{attribute 'GeneratedUsingTerminal: APS4322-7000-0017'}
{attribute addProperty BoxType "APS4322-7000-0017"}
{attribute addProperty Id "StatusWordAT %I*UINT2Current_D_0X0AT %I*INT2Current_D_0X1AT %I*INT2Current_D_0X2AT %I*INT2Current_D_0Y0AT %I*INT2Current_D_0Y1AT %I*INT2Current_D_0Y2AT %I*INT2Current_D_1X0AT %I*INT2Current_D_1X1AT %I*INT2Current_D_1X2AT %I*INT2Current_D_1Y0AT %I*INT2Current_D_1Y1AT %I*INT2Current_D_1Y2AT %I*INT2Current_D_2X0AT %I*INT2Current_D_2X1AT %I*INT2Current_D_2X2AT %I*INT2Current_D_2Y0AT %I*INT2Current_D_2Y1AT %I*INT2Current_D_2Y2AT %I*INT2Current_D_3X0AT %I*INT2Current_D_3X1AT %I*INT2Current_D_3X2AT %I*INT2Current_D_3Y0AT %I*INT2Current_D_3Y1AT %I*INT2Current_D_3Y2AT %I*INT2Current_Q_0X0AT %I*INT2Current_Q_0X1AT %I*INT2Current_Q_0X2AT %I*INT2Current_Q_0Y0AT %I*INT2Current_Q_0Y1AT %I*INT2Current_Q_0Y2AT %I*INT2Current_Q_1X0AT %I*INT2Current_Q_1X1AT %I*INT2Current_Q_1X2AT %I*INT2Current_Q_1Y0AT %I*INT2Current_Q_1Y1AT %I*INT2Current_Q_1Y2AT %I*INT2Current_Q_2X0AT %I*INT2Current_Q_2X1AT %I*INT2Current_Q_2X2AT %I*INT2Current_Q_2Y0AT %I*INT2Current_Q_2Y1AT %I*INT2Current_Q_2Y2AT %I*INT2Current_Q_3X0AT %I*INT2Current_Q_3X1AT %I*INT2Current_Q_3X2AT %I*INT2Current_Q_3Y0AT %I*INT2Current_Q_3Y1AT %I*INT2Current_Q_3Y2AT %I*INT2"}
{attribute addProperty CRC "1192874203"}
{attribute addProperty Size "98"}
TYPE APS_Inputs_4719D0DB :
STRUCT
	{attribute addProperty Name "StatusWord"}
	StatusWord AT %I* : UINT;
	{attribute addProperty Name "Current_D_0X0"}
	Current_D_0X0 AT %I* : INT;
	{attribute addProperty Name "Current_D_0X1"}
	Current_D_0X1 AT %I* : INT;
	{attribute addProperty Name "Current_D_0X2"}
	Current_D_0X2 AT %I* : INT;
	{attribute addProperty Name "Current_D_0Y0"}
	Current_D_0Y0 AT %I* : INT;
	{attribute addProperty Name "Current_D_0Y1"}
	Current_D_0Y1 AT %I* : INT;
	{attribute addProperty Name "Current_D_0Y2"}
	Current_D_0Y2 AT %I* : INT;
	{attribute addProperty Name "Current_D_1X0"}
	Current_D_1X0 AT %I* : INT;
	{attribute addProperty Name "Current_D_1X1"}
	Current_D_1X1 AT %I* : INT;
	{attribute addProperty Name "Current_D_1X2"}
	Current_D_1X2 AT %I* : INT;
	{attribute addProperty Name "Current_D_1Y0"}
	Current_D_1Y0 AT %I* : INT;
	{attribute addProperty Name "Current_D_1Y1"}
	Current_D_1Y1 AT %I* : INT;
	{attribute addProperty Name "Current_D_1Y2"}
	Current_D_1Y2 AT %I* : INT;
	{attribute addProperty Name "Current_D_2X0"}
	Current_D_2X0 AT %I* : INT;
	{attribute addProperty Name "Current_D_2X1"}
	Current_D_2X1 AT %I* : INT;
	{attribute addProperty Name "Current_D_2X2"}
	Current_D_2X2 AT %I* : INT;
	{attribute addProperty Name "Current_D_2Y0"}
	Current_D_2Y0 AT %I* : INT;
	{attribute addProperty Name "Current_D_2Y1"}
	Current_D_2Y1 AT %I* : INT;
	{attribute addProperty Name "Current_D_2Y2"}
	Current_D_2Y2 AT %I* : INT;
	{attribute addProperty Name "Current_D_3X0"}
	Current_D_3X0 AT %I* : INT;
	{attribute addProperty Name "Current_D_3X1"}
	Current_D_3X1 AT %I* : INT;
	{attribute addProperty Name "Current_D_3X2"}
	Current_D_3X2 AT %I* : INT;
	{attribute addProperty Name "Current_D_3Y0"}
	Current_D_3Y0 AT %I* : INT;
	{attribute addProperty Name "Current_D_3Y1"}
	Current_D_3Y1 AT %I* : INT;
	{attribute addProperty Name "Current_D_3Y2"}
	Current_D_3Y2 AT %I* : INT;
	{attribute addProperty Name "Current_Q_0X0"}
	Current_Q_0X0 AT %I* : INT;
	{attribute addProperty Name "Current_Q_0X1"}
	Current_Q_0X1 AT %I* : INT;
	{attribute addProperty Name "Current_Q_0X2"}
	Current_Q_0X2 AT %I* : INT;
	{attribute addProperty Name "Current_Q_0Y0"}
	Current_Q_0Y0 AT %I* : INT;
	{attribute addProperty Name "Current_Q_0Y1"}
	Current_Q_0Y1 AT %I* : INT;
	{attribute addProperty Name "Current_Q_0Y2"}
	Current_Q_0Y2 AT %I* : INT;
	{attribute addProperty Name "Current_Q_1X0"}
	Current_Q_1X0 AT %I* : INT;
	{attribute addProperty Name "Current_Q_1X1"}
	Current_Q_1X1 AT %I* : INT;
	{attribute addProperty Name "Current_Q_1X2"}
	Current_Q_1X2 AT %I* : INT;
	{attribute addProperty Name "Current_Q_1Y0"}
	Current_Q_1Y0 AT %I* : INT;
	{attribute addProperty Name "Current_Q_1Y1"}
	Current_Q_1Y1 AT %I* : INT;
	{attribute addProperty Name "Current_Q_1Y2"}
	Current_Q_1Y2 AT %I* : INT;
	{attribute addProperty Name "Current_Q_2X0"}
	Current_Q_2X0 AT %I* : INT;
	{attribute addProperty Name "Current_Q_2X1"}
	Current_Q_2X1 AT %I* : INT;
	{attribute addProperty Name "Current_Q_2X2"}
	Current_Q_2X2 AT %I* : INT;
	{attribute addProperty Name "Current_Q_2Y0"}
	Current_Q_2Y0 AT %I* : INT;
	{attribute addProperty Name "Current_Q_2Y1"}
	Current_Q_2Y1 AT %I* : INT;
	{attribute addProperty Name "Current_Q_2Y2"}
	Current_Q_2Y2 AT %I* : INT;
	{attribute addProperty Name "Current_Q_3X0"}
	Current_Q_3X0 AT %I* : INT;
	{attribute addProperty Name "Current_Q_3X1"}
	Current_Q_3X1 AT %I* : INT;
	{attribute addProperty Name "Current_Q_3X2"}
	Current_Q_3X2 AT %I* : INT;
	{attribute addProperty Name "Current_Q_3Y0"}
	Current_Q_3Y0 AT %I* : INT;
	{attribute addProperty Name "Current_Q_3Y1"}
	Current_Q_3Y1 AT %I* : INT;
	{attribute addProperty Name "Current_Q_3Y2"}
	Current_Q_3Y2 AT %I* : INT;
END_STRUCT
END_TYPE

(* stored: Version 1.2.0.0, ProductVersion 3.1.4024.9
   DUT APS_Inputs_4719D0DB: Id {53c2e460-37d0-4f86-b05a-b06d48f1e1bb} *)
